PROGRAM MAIN
VAR
	fbPlantControl : FB_PlantControl;
	Ctrl_data_Plant : Udt_PlantControl_Out;
	
	fbRunApp : FB_runApp;
END_VAR
VAR_IN_OUT
	
END_VAR


fbPlantControl(
	//Set up variables to IO here
	Auto_In := FIO.bAuto,
	Manual_In := FIO.bManual,
	
	Start_In := FIO.bStart,
	Stop_In := FIO.bStop,
	EmgStop_In := FIO.bEmgStop,
	Reset_In := FIO.bReset,
	
	Startet_Out => FIO.bGreenLight,
	Stopped_Out => FIO.bYellowLight,
	EmgStopped_Out => FIO.bRedLight,

	Ctrl_Plant := Ctrl_data_Plant
	);
	
IF fbPlantControl.Auto_Out THEN
	fbRunApp();
END_IF

END_PROGRAM

(* stored: Version 1.1.0.1, ProductVersion 3.1.4024.13
   POU MAIN: Id {afe816a1-7fba-460f-a8ae-1ac654733542}, SpecialFunc None *)
